FUNCTION_BLOCK MotorVsBase_HMI (* Service Interface Function Block Type *)
  (* Standard: 61499-2 *)
  (* Version 1.0.1, 2/5/2024, ApplicationLibDevTeam, Schneider Electric, First Version *)
  PACKAGE Main;
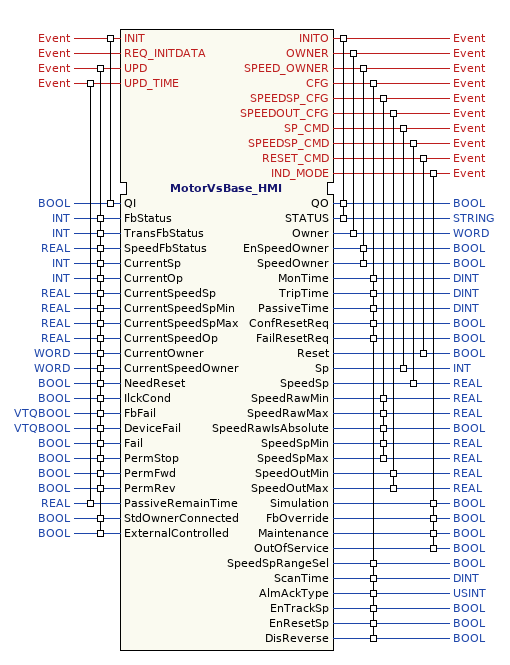
  EVENT_INPUT
    INIT WITH QI;
    REQ_INITDATA; (* Request to initialize data *)
    UPD WITH FbStatus, TransFbStatus, SpeedFbStatus, CurrentSp, CurrentOp, CurrentSpeedSp, CurrentSpeedOp, CurrentOwner, NeedReset, IlckCond, FbFail, DeviceFail, Fail, PermStop, PermFwd, PermRev, StdOwnerConnected, CurrentSpeedOwner, CurrentSpeedSpMin, CurrentSpeedSpMax, ExternalControlled; (* Update data to supervision *)
    UPD_TIME WITH PassiveRemainTime; (* Update time variables *)
  END_EVENT
  EVENT_OUTPUT
    INITO WITH QO, STATUS;
    OWNER WITH Owner; (* Request for owner change *)
    SPEED_OWNER WITH EnSpeedOwner, SpeedOwner; (* Request for speed owner change *)
    CFG WITH MonTime, TripTime, PassiveTime, ConfResetReq, FailResetReq, ScanTime, AlmAckType, EnTrackSp, EnResetSp, DisReverse, SpeedSpRangeSel; (* Request for new parameter *)
    SPEEDSP_CFG WITH SpeedRawMin, SpeedRawMax, SpeedRawIsAbsolute, SpeedSpMin, SpeedSpMax; (* Request for new speed setpoint parameter *)
    SPEEDOUT_CFG WITH SpeedOutMin, SpeedOutMax; (* Request for new speed output parameter *)
    SP_CMD WITH Sp; (* Request for new operator setpoint *)
    SPEEDSP_CMD WITH SpeedSp; (* Request for new operator speed setpoint *)
    RESET_CMD WITH Reset; (* Request to reset device *)
    IND_MODE WITH Simulation, FbOverride, Maintenance, OutOfService; (* Request for new operational modes *)
  END_EVENT
  VAR_INPUT
    QI : BOOL;
    FbStatus : INT; (* Device state(0 = stopped, 1= Running Forward, 2 = Running Reverse) *) {SET_ATTRIBUTE(Runtime.Archive.Counters, AbsoluteValues=False)} {SET_ATTRIBUTE(Runtime.Archive.Id, 1)} {SET_ATTRIBUTE(Runtime.History.Depth, 100)} {SET_ATTRIBUTE(Runtime.History.SmoothTime, 60000)} {SET_ATTRIBUTE(Runtime.History.SmoothValue, 1)}
    TransFbStatus : INT; (* Device transition state( 0 = stopped, 1= Running Forward, 2 = Running Reverse, 5 = Starting , 6 = Stopping and 253 = Unknown) *) {SET_ATTRIBUTE(Runtime.Archive.Counters, AbsoluteValues=False)} {SET_ATTRIBUTE(Runtime.Archive.Id, 1)} {SET_ATTRIBUTE(Runtime.History.Depth, 100)} {SET_ATTRIBUTE(Runtime.History.SmoothTime, 60000)} {SET_ATTRIBUTE(Runtime.History.SmoothValue, 1)}
    SpeedFbStatus : REAL; (* Speed feedback *) {SET_ATTRIBUTE(Runtime.Archive.Counters, )} {SET_ATTRIBUTE(Runtime.Archive.Id, 0)} {SET_ATTRIBUTE(Runtime.History.Depth, 0)} {SET_ATTRIBUTE(Runtime.History.SmoothTime, 0)} {SET_ATTRIBUTE(Runtime.History.SmoothValue, 0)}
    CurrentSp : INT; (* Current value of the direction setpoint *) {SET_ATTRIBUTE(Runtime.Archive.Counters, AbsoluteValues=False)} {SET_ATTRIBUTE(Runtime.Archive.Id, 1)} {SET_ATTRIBUTE(Runtime.History.Depth, 100)} {SET_ATTRIBUTE(Runtime.History.SmoothTime, 60000)} {SET_ATTRIBUTE(Runtime.History.SmoothValue, 1)}
    CurrentOp : INT; (* Current value of the output *) {SET_ATTRIBUTE(Runtime.Archive.Counters, AbsoluteValues=False)} {SET_ATTRIBUTE(Runtime.Archive.Id, 1)} {SET_ATTRIBUTE(Runtime.History.Depth, 100)} {SET_ATTRIBUTE(Runtime.History.SmoothTime, 60000)} {SET_ATTRIBUTE(Runtime.History.SmoothValue, 1)}
    CurrentSpeedSp : REAL; (* Current speed setpoint *)
    CurrentSpeedSpMin : REAL; (* Current speed minimum range *)
    CurrentSpeedSpMax : REAL; (* Current speed maximum range *)
    CurrentSpeedOp : REAL; (* Current speed output *)
    CurrentOwner : WORD; (* Current owner status *)
    CurrentSpeedOwner : WORD; (* Current speed owner status *)
    NeedReset : BOOL; (* 1 = Device need reset *)
    IlckCond : BOOL; (* 1 = Interlock Active *)
    FbFail : VTQBOOL; (* 1 = Feedback fail alarm status active *)
    DeviceFail : VTQBOOL; (* 1 = Device fail alarm status active *)
    Fail : BOOL; (* 1 = Fail Active *)
    PermStop : BOOL; (* 1 = Stop permission available *)
    PermFwd : BOOL; (* 1 = Forward start permission available *)
    PermRev : BOOL; (* 1 = Reverse start permission available *)
    PassiveRemainTime : REAL; (* Remaining time during direction change *)
    StdOwnerConnected : BOOL; (* 1= External owner Connected *)
    ExternalControlled : BOOL; (* 1 = Device is externally controlled *)
  END_VAR
  VAR_OUTPUT
    QO : BOOL; (* Event Output Qualifier *)
    STATUS : STRING; (* Service Status *)
    Owner : WORD; (* Requested Owner (16#10 = Operator, 16#8 = Program remote) *)
    EnSpeedOwner : BOOL; (* 1 = Enable speed owner *)
    SpeedOwner : BOOL; (* Speed owner is: 1= Operator, 0 = Program *)
    MonTime : DINT; (* Feedback monitoring time *)
    TripTime : DINT; (* Feedback trip time *)
    PassiveTime : DINT; (* Direction switch time *)
    ConfResetReq : BOOL; (* 1= Need reset on confirmation mismatch *)
    FailResetReq : BOOL; (* 1 = Need reset on device detected failure *)
    Reset : BOOL; (* 1 = Reset request from supervision *)
    Sp : INT; (* New direction setpoint from the supervision *)
    SpeedSp : REAL; (* New speed setpoint from the supervision *)
    SpeedRawMin : REAL; (* Minimum range of speed raw value *)
    SpeedRawMax : REAL; (* Maximum range of speed raw value *)
    SpeedRawIsAbsolute : BOOL; (* 1 = Absolute value of speed raw value will be considered for operation *)
    SpeedSpMin : REAL; (* Minimum range of speed setpoint *)
    SpeedSpMax : REAL; (* Maximum range of speed setpoint *)
    SpeedOutMin : REAL; (* Minimum range of speed ouput *)
    SpeedOutMax : REAL; (* Maximum range of speed output *)
    Simulation : BOOL; (* 1 = Enable device in simulation *)
    FbOverride : BOOL; (* 1 = Enable device in override mode *)
    Maintenance : BOOL; (* 1 = Enable device in maintenance mode *)
    OutOfService : BOOL; (* 1 = Out of Service Mode selected *)
    SpeedSpRangeSel : BOOL; (* SpeedSp range selection; 0 = Selection from HMI, 1 = Selection from service extension adapter/input pins *)
    ScanTime : DINT; (* Alarm holding time *)
    AlmAckType : USINT; (* 0=Not ackable; 1=Ack deletes; 2=Came has to be acked; 3=Came and gone have to be acked; 4=Pair has to be acked *)
    EnTrackSp : BOOL; (* 1= Enable the tracking of Interlock setpoint *)
    EnResetSp : BOOL; (* 1= Enable Reset Setpoint *)
    DisReverse : BOOL; (* Device is: 1 = Unidirectional, 0 = Bidirectional *)
  END_VAR
  SERVICE /
    SEQUENCE 
    END_SEQUENCE
  END_SERVICE
END_FUNCTION_BLOCK
